// TIA Portal V16 export
// export: Created 2023-03-29T11:03:17.249399Z, ExportSetting WithDefaults, DisplayName Totally Integrated Automation Portal, DisplayVersion V16 Update 6, DisplayName TIA Portal Version Control Interface, DisplayVersion V16 Update 2, DisplayName TIA Portal Openness, DisplayVersion V16 Update 6, DisplayName STEP 7 Professional, DisplayVersion V16 Update 6, DisplayName STEP 7 Safety, DisplayVersion V16, DisplayName WinCC Advanced, DisplayVersion V16 Update 6
ORGANIZATION_BLOCK "Diagnostic error interrupt"   // OB82, LAD, DiagnosticErrorInterrupt
{ S7_Optimized_Access := 'TRUE' }
VERSION : 0.1
// stored: IsIECCheckEnabled false, SetENOAutomatically false
   VAR_INPUT
      IO_State : Word;   // IO state of the HW object
      LADDR : HW_ANY;   // Hardware identifier
      Channel : UInt;   // Channel number
      MultiError : Bool;   // =true if more than one error is present
   END_VAR
   VAR_TEMP
      RetVal_RD_SYS_T : Int;   // //Status of the instruction RD_SYS_T: Read time-of-day
   END_VAR
BEGIN

REGION Network 2 (SCL)
   "EX012_ErrorBuffer_OB82".OB82ErrorCounter := "EX012_ErrorBuffer_OB82".OB82ErrorCounter + 1;
   //ochrona przed przepełnieniem tabeli
   IF ("EX012_ErrorBuffer_OB82".OB82ErrorCounter > "CONST_BUFFER_OB82") THEN
     "EX012_ErrorBuffer_OB82".OB82ErrorCounter := 1;
   END_IF;
   //Wystąpił błąd czasu
   #RetVal_RD_SYS_T := RD_LOC_T(OUT => "EX012_ErrorBuffer_OB82".ErrorDataOB82["EX012_ErrorBuffer_OB82".OB82ErrorCounter].ErrorTimestamp);
   //Zapis błedu do buffora (ErrorBuffor)
   "EX012_ErrorBuffer_OB82".ErrorDataOB82["EX012_ErrorBuffer_OB82".OB82ErrorCounter].IO_State := #IO_State;
   "EX012_ErrorBuffer_OB82".ErrorDataOB82["EX012_ErrorBuffer_OB82".OB82ErrorCounter].LADDR := #LADDR;
   "EX012_ErrorBuffer_OB82".ErrorDataOB82["EX012_ErrorBuffer_OB82".OB82ErrorCounter].Channel := #Channel;
   "EX012_ErrorBuffer_OB82".ErrorDataOB82["EX012_ErrorBuffer_OB82".OB82ErrorCounter].MultiError := #MultiError;
END_REGION
END_ORGANIZATION_BLOCK
